FUNCTION_BLOCK Motor_Dosagem_HMI (* Service Interface Function Block Type *)
  (* Standard: 61499-2 *)
  (* Version 0.0, 1/22/2026, Schneider Electric, template *)
  PACKAGE Hidryco.HidrycoLib;
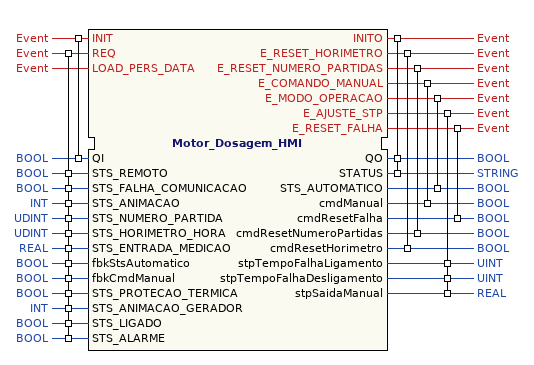
  EVENT_INPUT
    INIT WITH QI;
    REQ WITH STS_REMOTO, STS_ANIMACAO, STS_HORIMETRO_HORA, STS_ENTRADA_MEDICAO, fbkStsAutomatico, fbkCmdManual, STS_PROTECAO_TERMICA, STS_FALHA_COMUNICACAO, STS_NUMERO_PARTIDA, STS_ANIMACAO_GERADOR, STS_LIGADO, STS_ALARME;
    LOAD_PERS_DATA;
  END_EVENT
  EVENT_OUTPUT
    INITO WITH QO, STATUS;
    E_RESET_HORIMETRO WITH cmdResetHorimetro;
    E_RESET_NUMERO_PARTIDAS WITH cmdResetNumeroPartidas;
    E_COMANDO_MANUAL WITH cmdManual;
    E_MODO_OPERACAO WITH STS_AUTOMATICO;
    E_AJUSTE_STP WITH stpTempoFalhaLigamento, stpTempoFalhaDesligamento, stpSaidaManual;
    E_RESET_FALHA WITH cmdResetFalha;
  END_EVENT
  VAR_INPUT
    QI : BOOL;
    STS_REMOTO : BOOL;
    STS_FALHA_COMUNICACAO : BOOL;
    STS_ANIMACAO : INT;
    STS_NUMERO_PARTIDA : UDINT;
    STS_HORIMETRO_HORA : UDINT;
    STS_ENTRADA_MEDICAO : REAL;
    fbkStsAutomatico : BOOL;
    fbkCmdManual : BOOL;
    STS_PROTECAO_TERMICA : BOOL;
    STS_ANIMACAO_GERADOR : INT;
    STS_LIGADO : BOOL;
    STS_ALARME : BOOL;
  END_VAR
  VAR_OUTPUT
    QO : BOOL; (* Event Output Qualifier *)
    STATUS : STRING; (* Service Status *)
    STS_AUTOMATICO : BOOL; (* 0 - Manual, 1 - Automatico *)
    cmdManual : BOOL; (* 0 - Desligar, 1 - Ligar *)
    cmdResetFalha : BOOL;
    cmdResetNumeroPartidas : BOOL;
    cmdResetHorimetro : BOOL;
    stpTempoFalhaLigamento : UINT;
    stpTempoFalhaDesligamento : UINT;
    stpSaidaManual : REAL;
  END_VAR
  SERVICE /
    SEQUENCE 
    END_SEQUENCE
  END_SERVICE
END_FUNCTION_BLOCK
